ABB RobotStudio station: IRC5Sim_20230605-092405.rsstn

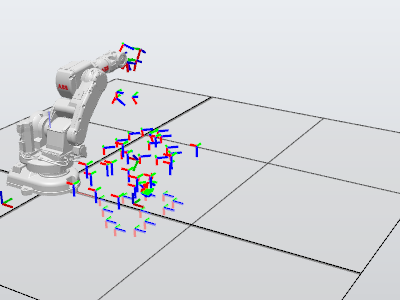
Station Station (saved by RobotStudio 22.3.10190.2)
Controller IRB140_6_81
  mechanical unit ROB_1: IRB140_6_81_C_03, 6 joints, base frame (0, 0, 0) mm
Layout (positions relative to the parent item):
  - IRB140_6_81_C_03 [mechanism, from Robots\IRB140_6_81_C_G_03.rslib] at (0, 0, 0) mm; joint values [1.5708, 0.6981, -0.7854, 0, 0, 0] (rad or m)
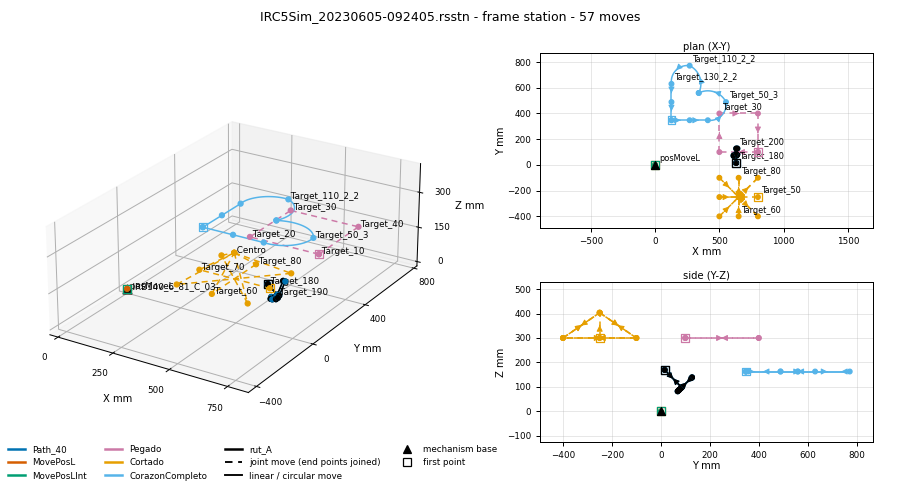
[picture p0: tool path of IRC5Sim_20230605-092405.rsstn in frame station, 57 of 73 moves have a stored position in this frame; points joined in program order, loops and branches not executed]
Targets, tools, work objects and paths stored in the station, written as RAPID:
! task T_ROB1
MODULE CalibData
  PERS tooldata ToolAJATCP:=[TRUE,[[71.4,0,67.85],[0.819152044,0,0.573576436,0]],[0.1,[0,0,1],[1,0,0,0],0,0,0]];
  TASK PERS wobjdata WOAJA:=[FALSE,TRUE,"",[[500,204.716,213.45],[0,0,-0.374478973,0.927235406]],[[0,0,0],[1,0,0,0]]];
  TASK PERS wobjdata MiMarcoDeCorazon:=[FALSE,TRUE,"",[[-120,100,70],[0.923879533,0,0,0.382683432]],[[0,0,93],[1,0,0,0]]];
  PERS tooldata TD_Hook:=[TRUE,[[68.38,0,60],[0.707106781,0.707106781,0,0]],[0.2,[28.798,-0.092,56.062],[1,0,0,0],0,0,0]];
  PERS tooldata TD_SuctionPad:=[TRUE,[[93.75,0,168.37],[0.970295726,0,0.241921896,0]],[0.2,[28.798,-0.092,56.062],[1,0,0,0],0,0,0]];
  PERS tooldata TD_SuctionPad2:=[TRUE,[[93.75,0,168.37],[0.970295726,0,0.241921896,0]],[0.2,[28.798,-0.092,56.062],[1,0,0,0],0,0,0]];
  TASK PERS wobjdata Workobject_1:=[FALSE,TRUE,"",[[-200,-850,260],[1,0,0,0]],[[475,140,0],[1,0,0,0]]];
  TASK PERS wobjdata Workobject_Balde_Piso:=[FALSE,TRUE,"",[[600,0,30],[1,0,0,0]],[[0,0,0],[1,0,0,0]]];
  PERS tooldata MyTool:=[TRUE,[[31.792631019,0,229.638935148],[0.945518576,0,0.325568154,0]],[1,[0,0,1],[1,0,0,0],0,0,0]];
  TASK PERS wobjdata Workobject_2:=[FALSE,TRUE,"",[[0,0,0],[1,0,0,0]],[[0,0,0],[1,0,0,0]]];
  TASK PERS wobjdata Workobject_C2:=[FALSE,TRUE,"",[[0,0,0],[1,0,0,0]],[[0,0,0],[1,0,0,0]]];
  TASK PERS wobjdata Workobject_C1:=[FALSE,TRUE,"",[[0,0,0],[1,0,0,0]],[[0,0,0],[1,0,0,0]]];
ENDMODULE

! task T_ROB1
MODULE Module1
  CONST jointtarget JointTarget_2:=[[0,50,-40,70,-50,-50],[9E+09,9E+09,9E+09,9E+09,9E+09,9E+09]];
  CONST jointtarget JointTarget_1:=[[0,20,-20,40,-20,-20],[9E+09,9E+09,9E+09,9E+09,9E+09,9E+09]];
  CONST jointtarget HomeP:=[[0,0,0,0,0,0],[9E+09,9E+09,9E+09,9E+09,9E+09,9E+09]];
  CONST jointtarget JointTarget_4:=[[90,40,-45,0,0,0],[9E+09,9E+09,9E+09,9E+09,9E+09,9E+09]];
  CONST robtarget Target_180:=[[-130.684278975,166.513773343,100.000300403],[-0.000000024,0.819152044,-0.573576437,-0.000000024],[0,1,-1,1],[9E+09,9E+09,9E+09,9E+09,9E+09,9E+09]];
  CONST robtarget Target_190:=[[-130.684278975,166.513780154,0.000300403],[0.000000024,-0.707106781,0.707106781,0.000000024],[0,1,-1,1],[9E+09,9E+09,9E+09,9E+09,9E+09,9E+09]];
  CONST robtarget Target_200:=[[-130.684278975,107.401152167,0.000296377],[0.000000024,-0.707106781,0.707106781,0.000000024],[0,1,-1,1],[9E+09,9E+09,9E+09,9E+09,9E+09,9E+09]];
  CONST robtarget Target_210:=[[-140.172333582,107.401152167,0.000296377],[0.000000024,-0.707106781,0.707106781,0.000000024],[0,1,-1,1],[9E+09,9E+09,9E+09,9E+09,9E+09,9E+09]];
  CONST robtarget Target_220:=[[-140.172333582,167.537670939,0.000300473],[0.000000024,0.819152044,-0.573576437,-0.000000024],[0,1,-1,1],[9E+09,9E+09,9E+09,9E+09,9E+09,9E+09]];
  CONST robtarget Target_230:=[[-138.363459862,177.588865478,0.000301158],[0.000000024,0.819152044,-0.573576437,-0.000000024],[0,1,-1,1],[9E+09,9E+09,9E+09,9E+09,9E+09,9E+09]];
  CONST robtarget Target_240:=[[-132.936838702,184.67077674,0.00030164],[0.000000024,0.819152044,-0.573576437,-0.000000024],[0,1,-1,1],[9E+09,9E+09,9E+09,9E+09,9E+09,9E+09]];
  CONST robtarget Target_250:=[[-118.807145869,188.971118037,0.000301932],[0.000000024,-0.707106781,0.707106781,0.000000024],[0,1,-1,1],[9E+09,9E+09,9E+09,9E+09,9E+09,9E+09]];
  CONST robtarget Target_260:=[[-111.23035406,188.561561724,0.000301905],[0.000000024,-0.707106781,0.707106781,0.000000024],[0,1,-1,1],[9E+09,9E+09,9E+09,9E+09,9E+09,9E+09]];
  CONST robtarget Target_270:=[[-110.820797746,180.779991758,0.000301375],[0.000000024,-0.707106781,0.707106781,0.000000024],[0,1,-1,1],[9E+09,9E+09,9E+09,9E+09,9E+09,9E+09]];
  CONST robtarget Target_280:=[[-123.482913787,180.353370597,0.000301346],[0.000000024,-0.707106781,0.707106781,0.000000024],[0,1,-1,1],[9E+09,9E+09,9E+09,9E+09,9E+09,9E+09]];
  CONST robtarget Target_290:=[[-129.882231193,172.605930324,0.000300819],[0.000000024,-0.707106781,0.707106781,0.000000024],[0,1,-1,1],[9E+09,9E+09,9E+09,9E+09,9E+09,9E+09]];
  CONST robtarget Target_300:=[[-130.684278975,166.513780154,0.000300403],[0.000000024,-0.707106781,0.707106781,0.000000024],[0,1,-1,1],[9E+09,9E+09,9E+09,9E+09,9E+09,9E+09]];
  CONST robtarget Target_310:=[[-130.684278975,166.513773343,100.000300403],[0.000000024,0.819152044,-0.573576437,-0.000000024],[0,1,-1,1],[9E+09,9E+09,9E+09,9E+09,9E+09,9E+09]];
  CONST jointtarget JointTarget_TL:=[[90,40,-45,0,0,0],[9E+09,9E+09,9E+09,9E+09,9E+09,9E+09]];
  CONST jointtarget JointTarget_TR:=[[-90,40,-45,0,0,0],[9E+09,9E+09,9E+09,9E+09,9E+09,9E+09]];
  VAR jointtarget myJointTarget:=[[0,0,0,0,0,0],[9E+09,9E+09,9E+09,9E+09,9E+09,9E+09]];
  VAR robtarget posMoveL:=[[0,0,0],[1,0,0,0],[0,0,0,0],[9E+09,9E+09,9E+09,9E+09,9E+09,9E+09]];
  CONST jointtarget HomeR:=[[0,0,0,0,30,0],[9E+09,9E+09,9E+09,9E+09,9E+09,9E+09]];
  CONST robtarget Target_10_3:=[[350,0,0],[0.707106781,0,0.707106781,0],[0,0,0,1],[9E+09,9E+09,9E+09,9E+09,9E+09,9E+09]];
  CONST robtarget Target_20_3:=[[450,-100,0],[0.707106781,0,0.707106781,0],[-1,-1,0,1],[9E+09,9E+09,9E+09,9E+09,9E+09,9E+09]];
  CONST robtarget Target_30_3:=[[550,-200,0],[0.707106781,0,0.707106781,0],[-1,-1,0,1],[9E+09,9E+09,9E+09,9E+09,9E+09,9E+09]];
  CONST robtarget Target_40_3:=[[650,-250,0],[0.707106781,0,0.707106781,0],[-1,-1,0,1],[9E+09,9E+09,9E+09,9E+09,9E+09,9E+09]];
  CONST robtarget Target_50_3:=[[750,-200,0],[0.707106781,0,0.707106781,0],[-1,-1,0,1],[9E+09,9E+09,9E+09,9E+09,9E+09,9E+09]];
  CONST robtarget Target_60_3:=[[750,-100,0],[0.707106781,0,0.707106781,0],[-1,-1,0,1],[9E+09,9E+09,9E+09,9E+09,9E+09,9E+09]];
  CONST robtarget Target_70_3:=[[650,0,0],[0.707106781,0,0.707106781,0],[0,0,0,1],[9E+09,9E+09,9E+09,9E+09,9E+09,9E+09]];
  CONST robtarget Target_80_2_2:=[[650,0,0],[0.707106781,0,0.707106781,0],[0,0,0,1],[9E+09,9E+09,9E+09,9E+09,9E+09,9E+09]];
  CONST robtarget Target_90_2_2:=[[750,100,0],[0.707106781,0,0.707106781,0],[-1,-1,0,1],[9E+09,9E+09,9E+09,9E+09,9E+09,9E+09]];
  CONST robtarget Target_110_2_2:=[[750,200,0],[0.707106781,0,0.707106781,0],[0,0,-1,1],[9E+09,9E+09,9E+09,9E+09,9E+09,9E+09]];
  CONST robtarget Target_120_2_2:=[[650,250,0],[0.707106781,0,0.707106781,0],[0,0,-1,1],[9E+09,9E+09,9E+09,9E+09,9E+09,9E+09]];
  CONST robtarget Target_130_2_2:=[[550,200,0],[0.707106781,0,0.707106781,0],[0,0,-1,1],[9E+09,9E+09,9E+09,9E+09,9E+09,9E+09]];
  CONST robtarget Target_140_2_2:=[[450,100,0],[0.707106781,0,0.707106781,0],[0,0,0,1],[9E+09,9E+09,9E+09,9E+09,9E+09,9E+09]];
  CONST robtarget Target_1010_2_2:=[[350,0,0],[0.707106781,0,0.707106781,0],[0,0,0,1],[9E+09,9E+09,9E+09,9E+09,9E+09,9E+09]];
  CONST robtarget home_2:=[[506.292,0,679.5],[0.5,0,0.866025404,0],[0,-2,-2,1],[9E+09,9E+09,9E+09,9E+09,9E+09,9E+09]];
  CONST robtarget Target_320:=[[238.002577223,458.002529699,842.500023251],[0.46193974,-0.331413514,0.800103175,0.19134176],[0,-3,-2,1],[9E+09,9E+09,9E+09,9E+09,9E+09,9E+09]];
  CONST robtarget Target_10:=[[800,100,300],[0,0,1,0],[0,0,0,0],[9E+09,9E+09,9E+09,9E+09,9E+09,9E+09]];
  CONST robtarget Target_20:=[[500,100,300],[0,0,1,0],[0,-1,0,0],[9E+09,9E+09,9E+09,9E+09,9E+09,9E+09]];
  CONST robtarget Target_30:=[[500,400,300],[0,0,1,0],[0,-1,0,0],[9E+09,9E+09,9E+09,9E+09,9E+09,9E+09]];
  CONST robtarget Target_40:=[[800,400,300],[0,0,1,0],[0,-1,0,0],[9E+09,9E+09,9E+09,9E+09,9E+09,9E+09]];
  CONST robtarget Target_50:=[[800,-250,300],[0,0,1,0],[0,0,0,0],[9E+09,9E+09,9E+09,9E+09,9E+09,9E+09]];
  CONST robtarget Target_70:=[[500,-250,300],[0,0,1,0],[-1,0,-1,0],[9E+09,9E+09,9E+09,9E+09,9E+09,9E+09]];
  CONST robtarget Centro:=[[650,-250,403.186020656],[0,0,1,0],[-1,0,-1,0],[9E+09,9E+09,9E+09,9E+09,9E+09,9E+09]];
  CONST robtarget Target_80:=[[650,-100,300],[0,0,1,0],[-1,0,-1,0],[9E+09,9E+09,9E+09,9E+09,9E+09,9E+09]];
  CONST robtarget Target_60:=[[650,-400,300],[0,0,1,0],[-1,0,-1,0],[9E+09,9E+09,9E+09,9E+09,9E+09,9E+09]];
  CONST robtarget Target_120:=[[800,-100,300],[0,0,1,0],[-1,0,-1,0],[9E+09,9E+09,9E+09,9E+09,9E+09,9E+09]];
  CONST robtarget Target_100:=[[500,-400,300],[0,0,1,0],[-1,0,-1,0],[9E+09,9E+09,9E+09,9E+09,9E+09,9E+09]];
  CONST robtarget Target_90:=[[800,-400,300],[0,0,1,0],[-1,0,-1,0],[9E+09,9E+09,9E+09,9E+09,9E+09,9E+09]];
  CONST robtarget Target_110:=[[500,-100,300],[0,0,1,0],[-1,0,-1,0],[9E+09,9E+09,9E+09,9E+09,9E+09,9E+09]];
  PROC main()
    ActualizarDatoPos;
    SetDO DO_IOT_01,1;
    WaitDI DI_IOT_02,1;
    WaitDI DI_IOT_01,1;
    WaitDI DI_IOT_02,1;
    SetDO DO_IOT_01,0;
    ToHomeP;
    ToHomeR;
    ToolQL;
    ToolQR;
    Security;
    MoveProcJInt;
    MovePosLInt;
    CortadoFull;
    CorazonCompleto;
    rut_A;
  ENDPROC
  PROC ToHome()
    MoveAbsJ JointTarget_2,v100,z10,ToolAJATCP\WObj:=WOAJA;
    ActualizarDatoPos;
    MoveAbsJ JointTarget_1,v100,z10,ToolAJATCP\WObj:=WOAJA;
    ActualizarDatoPos;
    MoveAbsJ HomeP,v100,z10,ToolAJATCP\WObj:=WOAJA;
  ENDPROC
  PROC Security()
    ActualizarDatoPos;
    MoveAbsJ HomeP,v100,z10,ToolAJATCP\WObj:=WOAJA;
    ActualizarDatoPos;
    MoveAbsJ JointTarget_1,v100,z10,ToolAJATCP\WObj:=WOAJA;
    ActualizarDatoPos;
    MoveAbsJ JointTarget_2,v100,z10,ToolAJATCP\WObj:=WOAJA;
  ENDPROC
  PROC ToolQ()
    MoveAbsJ HomeP,v100,z10,ToolAJATCP\WObj:=WOAJA;
    MoveAbsJ JointTarget_4,v100,z10,ToolAJATCP\WObj:=WOAJA;
  ENDPROC
  PROC Path_40()
    MoveL Target_180,v100,z10,ToolAJATCP\WObj:=WOAJA;
    MoveL Target_190,v100,z10,ToolAJATCP\WObj:=WOAJA;
    MoveL Target_200,v100,z10,ToolAJATCP\WObj:=WOAJA;
    MoveL Target_210,v100,z10,ToolAJATCP\WObj:=WOAJA;
    MoveL Target_220,v100,z10,ToolAJATCP\WObj:=WOAJA;
    MoveL Target_230,v100,z10,ToolAJATCP\WObj:=WOAJA;
    MoveL Target_240,v100,z10,ToolAJATCP\WObj:=WOAJA;
    MoveL Target_250,v100,z10,ToolAJATCP\WObj:=WOAJA;
    MoveL Target_260,v100,z10,ToolAJATCP\WObj:=WOAJA;
    MoveL Target_270,v100,z10,ToolAJATCP\WObj:=WOAJA;
    MoveL Target_280,v100,z10,ToolAJATCP\WObj:=WOAJA;
    MoveL Target_290,v100,z10,ToolAJATCP\WObj:=WOAJA;
    MoveL Target_300,v100,z10,ToolAJATCP\WObj:=WOAJA;
    MoveL Target_310,v100,z10,ToolAJATCP\WObj:=WOAJA;
  ENDPROC
  PROC ToolQL()
    MoveAbsJ HomeP,v200,z10,ToolAJATCP\WObj:=WOAJA;
    ActualizarDatoPos;
    MoveAbsJ JointTarget_TL,v100,z10,ToolAJATCP\WObj:=WOAJA;
  ENDPROC
  PROC ToolQR()
    ActualizarDatoPos;
    MoveAbsJ HomeP,v200,z10,ToolAJATCP\WObj:=WOAJA;
    ActualizarDatoPos;
    MoveAbsJ JointTarget_TR,v100,z10,ToolAJATCP\WObj:=WOAJA;
  ENDPROC
  PROC ActualizarDatoPos()
  ENDPROC
  PROC MovePosL()
    MoveL posMoveL,v50,z5,tool0\WObj:=wobj0;
  ENDPROC
  PROC ToHomeR()
    ActualizarDatoPos;
    MoveAbsJ HomeR,v200,z10,ToolAJATCP\WObj:=WOAJA;
  ENDPROC
  PROC ToHomeP()
    ActualizarDatoPos;
    MoveAbsJ HomeP,v200,z10,ToolAJATCP\WObj:=WOAJA;
  ENDPROC
  PROC MoveProcJ()
    MoveAbsJ myJointTarget,v100,z10,ToolAJATCP\WObj:=WOAJA;
  ENDPROC
  PROC MoveProcJInt()
    MoveAbsJ myJointTarget,v100,z10,ToolAJATCP\WObj:=WOAJA;
  ENDPROC
  PROC MovePosLInt()
    MoveL posMoveL,v50,z5,tool0\WObj:=wobj0;
  ENDPROC
  PROC CortadoFull()
    ToHomeR;
    Pegado;
    ToHomeR;
    Cortado;
    ToHomeR;
  ENDPROC
  PROC Pegado()
    MoveJ Target_10,v200,fine,MyTool\WObj:=Workobject_C1;
    MoveJ Target_20,v200,fine,MyTool\WObj:=Workobject_C1;
    MoveJ Target_30,v200,fine,MyTool\WObj:=Workobject_C1;
    MoveJ Target_40,v200,fine,MyTool\WObj:=Workobject_C1;
    MoveJ Target_10,v200,fine,MyTool\WObj:=Workobject_C1;
  ENDPROC
  PROC Cortado()
    MoveJ Target_50,v200,fine,MyTool\WObj:=Workobject_C2;
    MoveJ Target_70,v200,fine,MyTool\WObj:=Workobject_C2;
    MoveJ Centro,v200,fine,MyTool\WObj:=Workobject_C2;
    MoveJ Target_80,v200,fine,MyTool\WObj:=Workobject_C2;
    MoveJ Target_60,v200,fine,MyTool\WObj:=Workobject_C2;
    MoveJ Centro,v200,fine,MyTool\WObj:=Workobject_C2;
    MoveJ Target_120,v200,fine,MyTool\WObj:=Workobject_C2;
    MoveJ Target_100,v200,fine,MyTool\WObj:=Workobject_C2;
    MoveJ Centro,v200,fine,MyTool\WObj:=Workobject_C2;
    MoveJ Target_90,v200,fine,MyTool\WObj:=Workobject_C2;
    MoveJ Target_110,v200,fine,MyTool\WObj:=Workobject_C2;
    MoveJ Centro,v200,fine,MyTool\WObj:=Workobject_C2;
  ENDPROC
  PROC CorazonCompleto()
    MoveJ Target_10_3,v200,z5,tool0\WObj:=MiMarcoDeCorazon;
    MoveL Target_20_3,v200,z5,tool0\WObj:=MiMarcoDeCorazon;
    MoveL Target_30_3,v200,z5,tool0\WObj:=MiMarcoDeCorazon;
    MoveC Target_40_3,Target_50_3,v200,z5,tool0\WObj:=MiMarcoDeCorazon;
    MoveC Target_60_3,Target_70_3,v200,z5,tool0\WObj:=MiMarcoDeCorazon;
    MoveL Target_80_2_2,v200,z5,tool0\WObj:=MiMarcoDeCorazon;
    MoveC Target_90_2_2,Target_110_2_2,v200,z5,tool0\WObj:=MiMarcoDeCorazon;
    MoveC Target_120_2_2,Target_130_2_2,v200,z5,tool0\WObj:=MiMarcoDeCorazon;
    MoveL Target_140_2_2,v200,z5,tool0\WObj:=MiMarcoDeCorazon;
    MoveL Target_1010_2_2,v200,z5,tool0\WObj:=MiMarcoDeCorazon;
    ToHomeR;
  ENDPROC
  PROC rut_A()
    Security;
    MoveL Target_180,v100,z10,ToolAJATCP\WObj:=WOAJA;
    MoveL Target_190,v100,z10,ToolAJATCP\WObj:=WOAJA;
    MoveL Target_200,v100,z10,ToolAJATCP\WObj:=WOAJA;
    MoveL Target_210,v100,z10,ToolAJATCP\WObj:=WOAJA;
    MoveL Target_220,v100,z10,ToolAJATCP\WObj:=WOAJA;
    MoveL Target_230,v100,z10,ToolAJATCP\WObj:=WOAJA;
    MoveL Target_240,v100,z10,ToolAJATCP\WObj:=WOAJA;
    MoveL Target_250,v100,z10,ToolAJATCP\WObj:=WOAJA;
    MoveL Target_260,v100,z10,ToolAJATCP\WObj:=WOAJA;
    MoveL Target_270,v100,z10,ToolAJATCP\WObj:=WOAJA;
    MoveL Target_280,v100,z10,ToolAJATCP\WObj:=WOAJA;
    MoveL Target_290,v100,z10,ToolAJATCP\WObj:=WOAJA;
    MoveL Target_300,v100,z10,ToolAJATCP\WObj:=WOAJA;
    MoveL Target_310,v100,z10,ToolAJATCP\WObj:=WOAJA;
    ToHomeR;
  ENDPROC
ENDMODULE

